PROGRAM General
VAR
END_VAR

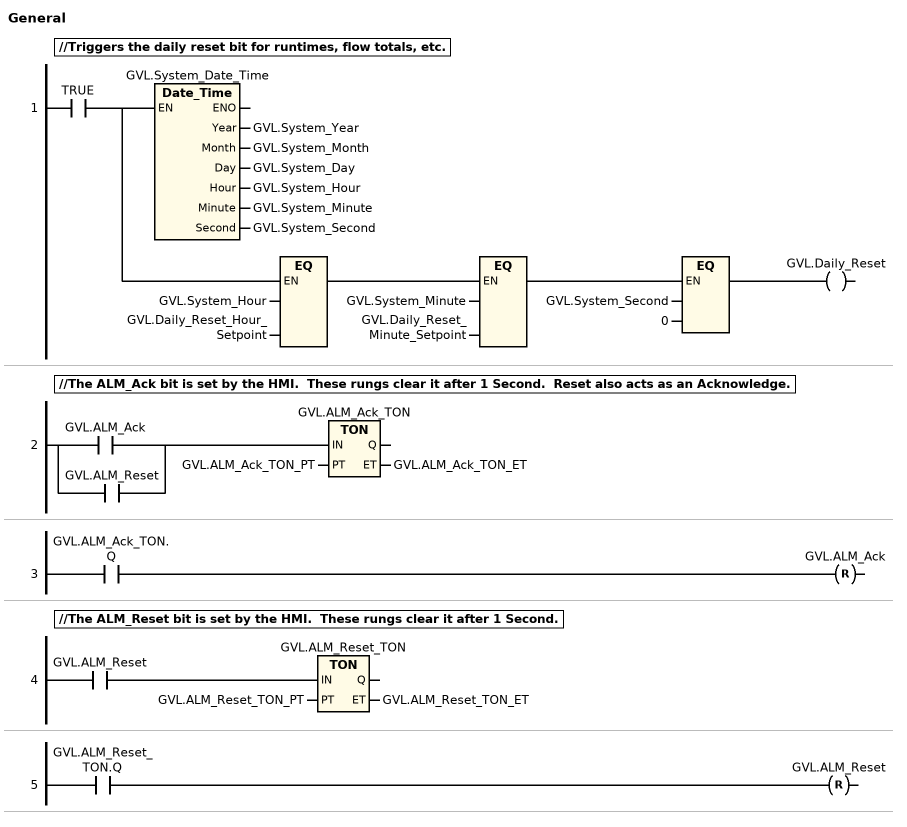
// NETWORK 1
// label: //Triggers the daily reset bit for runtimes, flow totals, etc.
GVL.System_Date_Time(
    Year => GVL.System_Year,
    Month => GVL.System_Month,
    Day => GVL.System_Day,
    Hour => GVL.System_Hour,
    Minute => GVL.System_Minute,
    Second => GVL.System_Second); // Date_Time
GVL.Daily_Reset := GVL.System_Hour = GVL.Daily_Reset_Hour_Setpoint AND GVL.System_Minute = GVL.Daily_Reset_Minute_Setpoint AND GVL.System_Second = 0;

// NETWORK 2
// label: //The ALM_Ack bit is set by the HMI.  These rungs clear it after 1 Second.  Reset also acts as an Acknowledge.
GVL.ALM_Ack_TON(IN := GVL.ALM_Ack OR GVL.ALM_Reset, PT := GVL.ALM_Ack_TON_PT, ET => GVL.ALM_Ack_TON_ET); // TON

// NETWORK 3
GVL.ALM_Ack R= GVL.ALM_Ack_TON.Q;

// NETWORK 4
// label: //The ALM_Reset bit is set by the HMI.  These rungs clear it after 1 Second.
GVL.ALM_Reset_TON(IN := GVL.ALM_Reset, PT := GVL.ALM_Reset_TON_PT, ET => GVL.ALM_Reset_TON_ET); // TON

// NETWORK 5
GVL.ALM_Reset R= GVL.ALM_Reset_TON.Q;

END_PROGRAM

(* stored: Version 1.1.0.1, ProductVersion 3.1.4024.12
   POU General: Id {afd5554c-a122-45cd-a612-91df6056dfdf}, SpecialFunc None *)
